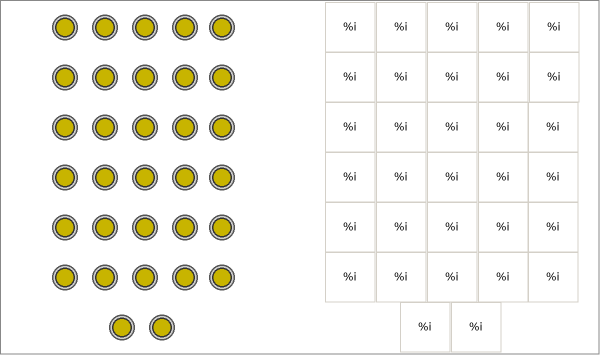
VISUALIZATION Set_Input  // 600x355
    Lamp1 (50,10 30x35), variable: HMI_Global.HMI_IN_Digital[0], style: Lamp-Lamp1-Yellow
    Lamp1 (90,10 30x35), variable: HMI_Global.HMI_IN_Digital[1], style: Lamp-Lamp1-Yellow
    Lamp1 (130,10 30x35), variable: HMI_Global.HMI_IN_Digital[2], style: Lamp-Lamp1-Yellow
    Lamp1 (170,10 30x35), variable: HMI_Global.HMI_IN_Digital[3], style: Lamp-Lamp1-Yellow
    Lamp1 (170,60 30x35), variable: HMI_Global.HMI_IN_Digital[8], style: Lamp-Lamp1-Yellow
    Lamp1 (50,60 30x35), variable: HMI_Global.HMI_IN_Digital[5], style: Lamp-Lamp1-Yellow
    Lamp1 (90,60 30x35), variable: HMI_Global.HMI_IN_Digital[6], style: Lamp-Lamp1-Yellow
    Lamp1 (130,60 30x35), variable: HMI_Global.HMI_IN_Digital[7], style: Lamp-Lamp1-Yellow
    Lamp1 (50,110 30x35), variable: HMI_Global.HMI_IN_Digital[10], style: Lamp-Lamp1-Yellow
    Lamp1 (170,110 30x35), variable: HMI_Global.HMI_IN_Digital[13], style: Lamp-Lamp1-Yellow
    Lamp1 (90,110 30x35), variable: HMI_Global.HMI_IN_Digital[11], style: Lamp-Lamp1-Yellow
    Lamp1 (130,110 30x35), variable: HMI_Global.HMI_IN_Digital[12], style: Lamp-Lamp1-Yellow
    Lamp1 (50,160 30x35), variable: HMI_Global.HMI_IN_Digital[15], style: Lamp-Lamp1-Yellow
    Lamp1 (90,160 30x35), variable: HMI_Global.HMI_IN_Digital[16], style: Lamp-Lamp1-Yellow
    Lamp1 (130,160 30x35), variable: HMI_Global.HMI_IN_Digital[17], style: Lamp-Lamp1-Yellow
    Lamp1 (170,160 30x35), variable: HMI_Global.HMI_IN_Digital[18], style: Lamp-Lamp1-Yellow
    Lamp1 (170,210 30x35), variable: HMI_Global.HMI_IN_Digital[23], style: Lamp-Lamp1-Yellow
    Lamp1 (50,210 30x35), variable: HMI_Global.HMI_IN_Digital[20], style: Lamp-Lamp1-Yellow
    Lamp1 (90,210 30x35), variable: HMI_Global.HMI_IN_Digital[21], style: Lamp-Lamp1-Yellow
    Lamp1 (130,210 30x35), variable: HMI_Global.HMI_IN_Digital[22], style: Lamp-Lamp1-Yellow
    Lamp1 (207,10 30x35), variable: HMI_Global.HMI_IN_Digital[4], style: Lamp-Lamp1-Yellow
    Lamp1 (207,60 30x35), variable: HMI_Global.HMI_IN_Digital[9], style: Lamp-Lamp1-Yellow
    Lamp1 (207,110 30x35), variable: HMI_Global.HMI_IN_Digital[14], style: Lamp-Lamp1-Yellow
    Lamp1 (207,160 30x35), variable: HMI_Global.HMI_IN_Digital[19], style: Lamp-Lamp1-Yellow
    Lamp1 (207,210 30x35), variable: HMI_Global.HMI_IN_Digital[24], style: Lamp-Lamp1-Yellow
    Lamp1 (170,260 30x35), variable: HMI_Global.HMI_IN_Digital[28], style: Lamp-Lamp1-Yellow
    Lamp1 (50,260 30x35), variable: HMI_Global.HMI_IN_Digital[25], style: Lamp-Lamp1-Yellow
    Lamp1 (90,260 30x35), variable: HMI_Global.HMI_IN_Digital[26], style: Lamp-Lamp1-Yellow
    Lamp1 (130,260 30x35), variable: HMI_Global.HMI_IN_Digital[27], style: Lamp-Lamp1-Yellow
    Lamp1 (207,260 30x35), variable: HMI_Global.HMI_IN_Digital[29], style: Lamp-Lamp1-Yellow
    Textfield (325,2 50x50), "%i", text variable: HMI_Global.HMI_IN_Analog[0]
        OnMouseDown: write the text variable via VisuDialogs.Numpad, min 0, max 1000
    Textfield (376,2 50x50), "%i", text variable: HMI_Global.HMI_IN_Analog[1]
        OnMouseDown: write the text variable via VisuDialogs.Numpad, min 0, max 1000
    Textfield (427,2 50x50), "%i", text variable: HMI_Global.HMI_IN_Analog[2]
        OnMouseDown: write the text variable via VisuDialogs.Numpad, min 0, max 1000
    Textfield (478,2 50x50), "%i", text variable: HMI_Global.HMI_IN_Analog[3]
        OnMouseDown: write the text variable via VisuDialogs.Numpad, min 0, max 1000
    Textfield (529,2 50x50), "%i", text variable: HMI_Global.HMI_IN_Analog[4]
        OnMouseDown: write the text variable via VisuDialogs.Numpad, min 0, max 1000
    Textfield (325,52 50x50), "%i", text variable: HMI_Global.HMI_IN_Analog[5]
        OnMouseDown: write the text variable via VisuDialogs.Numpad, min 0, max 1000
    Textfield (376,52 50x50), "%i", text variable: HMI_Global.HMI_IN_Analog[6]
        OnMouseDown: write the text variable via VisuDialogs.Numpad, min 0, max 1000
    Textfield (427,52 50x50), "%i", text variable: HMI_Global.HMI_IN_Analog[7]
        OnMouseDown: write the text variable via VisuDialogs.Numpad, min 0, max 1000
    Textfield (478,52 50x50), "%i", text variable: HMI_Global.HMI_IN_Analog[8]
        OnMouseDown: write the text variable via VisuDialogs.Numpad, min 0, max 1000
    Textfield (529,52 50x50), "%i", text variable: HMI_Global.HMI_IN_Analog[9]
        OnMouseDown: write the text variable via VisuDialogs.Numpad, min 0, max 1000
    Textfield (325,102 50x50), "%i", text variable: HMI_Global.HMI_IN_Analog[10]
        OnMouseDown: write the text variable via VisuDialogs.Numpad, min 0, max 1000
    Textfield (376,102 50x50), "%i", text variable: HMI_Global.HMI_IN_Analog[11]
        OnMouseDown: write the text variable via VisuDialogs.Numpad, min 0, max 1000
    Textfield (427,102 50x50), "%i", text variable: HMI_Global.HMI_IN_Analog[12]
        OnMouseDown: write the text variable via VisuDialogs.Numpad, min 0, max 1000
    Textfield (478,102 50x50), "%i", text variable: HMI_Global.HMI_IN_Analog[13]
        OnMouseDown: write the text variable via VisuDialogs.Numpad, min 0, max 1000
    Textfield (528,102 50x50), "%i", text variable: HMI_Global.HMI_IN_Analog[14]
        OnMouseDown: write the text variable via VisuDialogs.Numpad, min 0, max 1000
    Textfield (325,152 50x50), "%i", text variable: HMI_Global.HMI_IN_Analog[15]
        OnMouseDown: write the text variable via VisuDialogs.Numpad, min 0, max 1000
    Textfield (376,152 50x50), "%i", text variable: HMI_Global.HMI_IN_Analog[16]
        OnMouseDown: write the text variable via VisuDialogs.Numpad, min 0, max 1000
    Textfield (427,152 50x50), "%i", text variable: HMI_Global.HMI_IN_Analog[17]
        OnMouseDown: write the text variable via VisuDialogs.Numpad, min 0, max 1000
    Textfield (478,152 50x50), "%i", text variable: HMI_Global.HMI_IN_Analog[18]
        OnMouseDown: write the text variable via VisuDialogs.Numpad, min 0, max 1000
    Textfield (528,152 50x50), "%i", text variable: HMI_Global.HMI_IN_Analog[19]
        OnMouseDown: write the text variable via VisuDialogs.Numpad, min 0, max 1000
    Textfield (325,202 50x50), "%i", text variable: HMI_Global.HMI_IN_Analog[20]
        OnMouseDown: write the text variable via VisuDialogs.Numpad, min 0, max 1000
    Textfield (376,202 50x50), "%i", text variable: HMI_Global.HMI_IN_Analog[21]
        OnMouseDown: write the text variable via VisuDialogs.Numpad, min 0, max 1000
    Textfield (427,202 50x50), "%i", text variable: HMI_Global.HMI_IN_Analog[22]
        OnMouseDown: write the text variable via VisuDialogs.Numpad, min 0, max 1000
    Textfield (478,202 50x50), "%i", text variable: HMI_Global.HMI_IN_Analog[23]
        OnMouseDown: write the text variable via VisuDialogs.Numpad, min 0, max 1000
    Textfield (528,202 50x50), "%i", text variable: HMI_Global.HMI_IN_Analog[24]
        OnMouseDown: write the text variable via VisuDialogs.Numpad, min 0, max 1000
    Textfield (325,252 50x50), "%i", text variable: HMI_Global.HMI_IN_Analog[25]
        OnMouseDown: write the text variable via VisuDialogs.Numpad, min 0, max 1000
    Textfield (376,252 50x50), "%i", text variable: HMI_Global.HMI_IN_Analog[26]
        OnMouseDown: write the text variable via VisuDialogs.Numpad, min 0, max 1000
    Textfield (427,252 50x50), "%i", text variable: HMI_Global.HMI_IN_Analog[27]
        OnMouseDown: write the text variable via VisuDialogs.Numpad, min 0, max 1000
    Textfield (478,252 50x50), "%i", text variable: HMI_Global.HMI_IN_Analog[28]
        OnMouseDown: write the text variable via VisuDialogs.Numpad, min 0, max 1000
    Textfield (528,252 50x50), "%i", text variable: HMI_Global.HMI_IN_Analog[29]
        OnMouseDown: write the text variable via VisuDialogs.Numpad, min 0, max 1000
    Textfield (400,302 50x50), "%i", text variable: HMI_Global.HMI_IN_Analog[30]
        OnMouseDown: write the text variable via VisuDialogs.Numpad, min 0, max 1000
    Textfield (451,302 50x50), "%i", text variable: HMI_Global.HMI_IN_Analog[31]
        OnMouseDown: write the text variable via VisuDialogs.Numpad, min 0, max 1000
    Lamp1 (107,310 30x35), variable: HMI_Global.HMI_IN_Digital[30], style: Lamp-Lamp1-Yellow
    Lamp1 (147,310 30x35), variable: HMI_Global.HMI_IN_Digital[31], style: Lamp-Lamp1-Yellow
END_VISUALIZATION

(* stored: Version 1.1.0.1, ProductVersion 3.1.4024.12
   Visu Set_Input: Id {abdc5e98-c19f-4448-a849-6cde96c8c179} *)
